FUNCTION FC_GetLocalHostName : T_MaxString	// Returns the local host name

FC_GetLocalHostName := IING.localHostName;

END_FUNCTION

(* stored: Version 1.1.0.1, ProductVersion 3.1.4026.18
   POU FC_GetLocalHostName: Id {004f4cfb-894b-4bd7-946a-8b82e5ef7059}, SpecialFunc None *)
